# EPICS autosave request: stdApp/Db/timer.req
$(P)timer$(N):preset
$(P)timer$(N):update.SCAN
$(P)timer$(N):doStop.FLNK
